// TIA Portal project "hardware_interrupt" (V18)

(* hardware
DEVICE "S7-1200 station_1"  S7-1200 Station
   slot 0: "Rack_0"  S7-1200 Rack  Rack  V1.0
   slot 1: "PLC_1"  CPU 1214C DC/DC/DC  6ES7 214-1AG40-0XB0  V4.6
*)

// ===== PLC "PLC_1"  CPU 1214C DC/DC/DC =====

VAR_GLOBAL   // PLC tag table "Default tag table"
   "Tag_1" AT %Q0.1 : Bool;
   "Tag_2" AT %Q0.2 : Bool;
   "Tag_3" AT %Q0.3 : Bool;
   "Tag_4" AT %Q0.4 : Bool;
   "Tag_5" AT %MW0 : Int;
   "Tag_6" AT %MW4 : Int;
END_VAR

ORGANIZATION_BLOCK "Main"   // OB1, LAD, ProgramCycle
TITLE = "Main Program Sweep (Cycle)"
{ S7_Optimized_Access := 'TRUE' }
VERSION : 0.1
   VAR_INPUT
      Initial_Call : Bool;   // Initial call of this OB
      Remanence : Bool;   // =True, if remanent data are available
   END_VAR
BEGIN

REGION Network 1
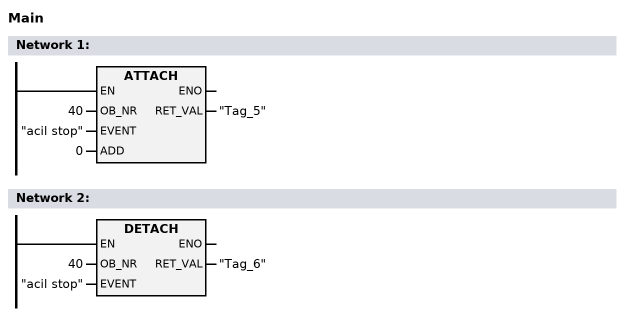
   "Tag_5" := ATTACH(OB_NR := 40, EVENT := "acil stop", ADD := 0);
END_REGION

REGION Network 2
   "Tag_6" := DETACH(OB_NR := 40, EVENT := "acil stop");
END_REGION
END_ORGANIZATION_BLOCK

ORGANIZATION_BLOCK "Hardware interrupt"   // OB40, LAD, HWProcessInterrupt
{ S7_Optimized_Access := 'TRUE' }
VERSION : 0.1
   VAR_INPUT
      LADDR : Hw_Io;   // Hardware identifier
      USI : Word;   // User structure identifier
      IChannel : USInt;   // Interrupt channel number
      EventType : Byte;   // EventType
   END_VAR
BEGIN

REGION Network 1
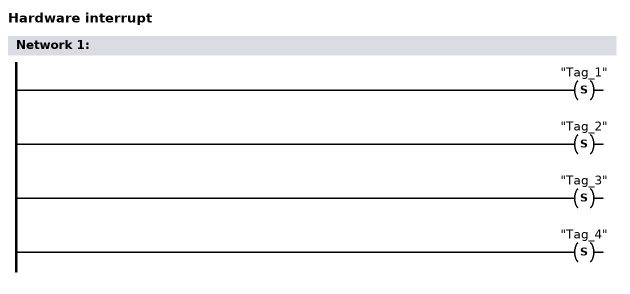
   RUNG wire#powerrail
      S_Coil( "Tag_1" )
   END_RUNG
   RUNG wire#powerrail
      S_Coil( "Tag_2" )
   END_RUNG
   RUNG wire#powerrail
      S_Coil( "Tag_3" )
   END_RUNG
   RUNG wire#powerrail
      S_Coil( "Tag_4" )
   END_RUNG
   // the same network as SCL:
   "Tag_1" := TRUE;
   "Tag_2" := TRUE;
   "Tag_3" := TRUE;
   "Tag_4" := TRUE;
END_REGION
END_ORGANIZATION_BLOCK